Omron Sysmac Studio project ExampleDataGenerator (Sysmac Studio 1.66.0.7, StandardProject)

# Controller Example: NX102-9000 version 1.64
Task PrimaryTask (priority 4, period or condition 2000): Generate

TYPE UintFlatArrayContainer : STRUCT
    array_1d : ARRAY[0..2] OF UINT;
    array_2d : ARRAY[0..2,0..2] OF UINT;
    array_3d : ARRAY[0..2,0..2,0..2] OF UINT;
END_STRUCT END_TYPE
TYPE ExampleStruct : STRUCT
    vel : LREAL;
    trq : LREAL;
    acc : LREAL;
    status_code : DWORD;
END_STRUCT END_TYPE
TYPE ExampleUnion : UNION
    status_flags : ARRAY[0..15] OF BOOL;
    segmented_status_codes : ARRAY[0..1] OF WORD;
    status_code : DWORD;
END_UNION END_TYPE
TYPE ExampleUnionContainer : STRUCT
    value : ExampleUnion;
END_STRUCT END_TYPE

PROGRAM Generate
VAR
    iFileWriteVar : FileWriteVar;
    UINT_SINGLE : UINT;
    UINT_ARRAY : UintFlatArrayContainer;
    EXAMPLE_STRUCT : ExampleStruct;
    EXAMPLE_UNION : ExampleUnionContainer;
END_VAR
VAR CONSTANT
    STATE_INIT : UINT := 0;
    STATE_CREATE_BIN : UINT := 20;
    STATE_FINALIZE : UINT := 900;
    STATE_DONE : UINT := 1000;
END_VAR
VAR
    WRITE_VAR_BASE_PATH : STRING[65];
    iState : UINT := 0;
    iReturnState : UINT;
    iVarIndex : UINT;
    iCurrentVarIndex : UINT;
    iVarName : STRING[256];
    iVarFilePath : STRING[65];
END_VAR
CASE iState OF
	0:
		iState := STATE_CREATE_BIN;
		
	// STATE_CREATE_BIN
	20:		
		WRITE_VAR_BASE_PATH := '/examplebin/';
		
		Inc(iState);
	21:		
		iVarIndex := 0;
		iCurrentVarIndex := 0;
		
		Inc(iState);
	22:
		iCurrentVarIndex := iVarIndex;
		CASE iVarIndex OF
			0:
				iVarName := 'uint_single';
				
				Clear(UINT_SINGLE);
				UINT_SINGLE := 1;
				
				Inc(iVarIndex);
			1:
				iVarName := 'uint_array';

				// Since it consists solely of UINT types, alignment and padding have no practical effect.
				Clear(UINT_ARRAY);
				UINT_ARRAY.array_1d[0] := 0; UINT_ARRAY.array_1d[1] := 1; UINT_ARRAY.array_1d[2] := 2;

				UINT_ARRAY.array_2d[0, 0] := 0; UINT_ARRAY.array_2d[0, 1] := 1; UINT_ARRAY.array_2d[0, 2] := 2;
				UINT_ARRAY.array_2d[1, 0] := 3; UINT_ARRAY.array_2d[1, 1] := 4; UINT_ARRAY.array_2d[1, 2] := 5;
				UINT_ARRAY.array_2d[2, 0] := 6; UINT_ARRAY.array_2d[2, 1] := 7; UINT_ARRAY.array_2d[2, 2] := 8;
				
				UINT_ARRAY.array_2d[0, 0] := 0; UINT_ARRAY.array_2d[0, 1] := 1; UINT_ARRAY.array_2d[0, 2] := 2;
				UINT_ARRAY.array_2d[1, 0] := 3; UINT_ARRAY.array_2d[1, 1] := 4; UINT_ARRAY.array_2d[1, 2] := 5;
				UINT_ARRAY.array_2d[2, 0] := 6; UINT_ARRAY.array_2d[2, 1] := 7; UINT_ARRAY.array_2d[2, 2] := 8;
				
				UINT_ARRAY.array_3d[0, 0, 0] := 0; UINT_ARRAY.array_3d[0, 0, 1] := 1; UINT_ARRAY.array_3d[0, 0, 2] := 2;
				UINT_ARRAY.array_3d[0, 1, 0] := 3; UINT_ARRAY.array_3d[0, 1, 1] := 4; UINT_ARRAY.array_3d[0, 1, 2] := 5;
				UINT_ARRAY.array_3d[0, 2, 0] := 6; UINT_ARRAY.array_3d[0, 2, 1] := 7; UINT_ARRAY.array_3d[0, 2, 2] := 8;

				UINT_ARRAY.array_3d[1, 0, 0] := 9; UINT_ARRAY.array_3d[1, 0, 1] := 10; UINT_ARRAY.array_3d[1, 0, 2] := 11;
				UINT_ARRAY.array_3d[1, 1, 0] := 12; UINT_ARRAY.array_3d[1, 1, 1] := 13; UINT_ARRAY.array_3d[1, 1, 2] := 14;
				UINT_ARRAY.array_3d[1, 2, 0] := 15; UINT_ARRAY.array_3d[1, 2, 1] := 16; UINT_ARRAY.array_3d[1, 2, 2] := 17;

				UINT_ARRAY.array_3d[2, 0, 0] := 18; UINT_ARRAY.array_3d[2, 0, 1] := 19; UINT_ARRAY.array_3d[2, 0, 2] := 20;
				UINT_ARRAY.array_3d[2, 1, 0] := 21; UINT_ARRAY.array_3d[2, 1, 1] := 22; UINT_ARRAY.array_3d[2, 1, 2] := 23;
				UINT_ARRAY.array_3d[2, 2, 0] := 24; UINT_ARRAY.array_3d[2, 2, 1] := 25; UINT_ARRAY.array_3d[2, 2, 2] := 26;

				Inc(iVarIndex);
			2:
				iVarName := 'example_struct';
				
				Clear(EXAMPLE_STRUCT);
				EXAMPLE_STRUCT.acc := 5.5;
				EXAMPLE_STRUCT.trq := 11.1;
				EXAMPLE_STRUCT.vel := 3.7;
				EXAMPLE_STRUCT.status_code := DWORD#16#0080_000F;
				
				Inc(iVarIndex);

			3:
				iVarName := 'example_union';

				// Since it is defined as a single-field structure and used as a standalone variable,
				// there is no practical impact from alignment or padding.
				Clear(EXAMPLE_UNION);
				EXAMPLE_UNION.value.status_code := DWORD#2#10000000_01000000_00100000_00010000;
				
				Inc(iVarIndex);
		ELSE
				iVarIndex := 1000;			
		END_CASE;
		
		IF iVarIndex < 1000 THEN		
			Inc(iState);
		ELSE
			iState := iState + 7;
		END_IF;
	23:
		iFileWriteVar(Execute:=FALSE, WriteVar:=iCurrentVarIndex);
		
		iVarFilePath := CONCAT(WRITE_VAR_BASE_PATH, iVarName, '.bin');
		iFileWriteVar.FileName := iVarFilePath;
		iFileWriteVar.OverWrite := TRUE;
		
		Inc(iState);
	24:
		CASE iCurrentVarIndex OF
			0: iFileWriteVar(Execute:=TRUE, WriteVar:=UINT_SINGLE);
			1: iFileWriteVar(Execute:=TRUE, WriteVar:=UINT_ARRAY);
			2: iFileWriteVar(Execute:=TRUE, WriteVar:=EXAMPLE_STRUCT);
			3: iFileWriteVar(Execute:=TRUE, WriteVar:=EXAMPLE_UNION);
		ELSE
			Inc(iState);
		END_CASE;
		
		IF iFileWriteVar.Done THEN
			iState := iState - 2;
		END_IF;
	29:
		iState := STATE_FINALIZE;

	// STATE_FINALIZE
	900:		
		iState := iState + 9;
	909:
		iState := STATE_DONE;
	
	// STATE_DONE
	1000:
		Inc(iState);
END_CASE;
END_PROGRAM